// TIA Portal V17 export
// export: Created 2025-03-10T13:11:51.2223995Z, ExportSetting WithDefaults, DisplayName Totally Integrated Automation Portal, DisplayVersion V17 Update 8, DisplayName TIA Portal Openness, DisplayVersion V17 Update 8, DisplayName TIA Portal Version Control Interface, DisplayVersion V17, DisplayName SINAMICS Startdrive Advanced, DisplayVersion V17 SP2, DisplayName SINAMICS Startdrive G110M, G120, G120C, G120D, G120P, G115D, DisplayVersion V17 SP2, DisplayName SINAMICS Startdrive G130, G150, S120, S150, SINAMICS MV, S210, DisplayVersion V17 SP2, DisplayName STEP 7 Professional, DisplayVersion V17 Update 8, DisplayName SINUMERIK ONE STEP 7 Toolbox, DisplayVersion V17 Update 12, DisplayName SINUMERIK 840D sl STEP 7 Toolbox, DisplayVersion V17 Update 12, DisplayName STEP 7 Safety, DisplayVersion V17 Update 6, DisplayName WinCC Advanced, DisplayVersion V17 Update 8
VAR_GLOBAL   // PLC tag table "TAGS_IO_FIXTURES_UNIT_03"
   "/////MEASURING_UNIT/////" AT %M4500.0 : Bool;
   UMEAS_PUSHER_LCT_Q AT %M4500.1 : Bool;   // MEASURING UNIT LOCATE PUSHER OUTPUT
   UMEAS_PUSHER_RTN_Q AT %M4500.2 : Bool;   // MEASURING UNIT RETURN PUSHER OUTPUT
   UMEAS_PUSHER_UNLOCK_Q AT %M4500.3 : Bool;   // MEASURING UNIT UNLOCK PUSHER OUTPUT
   UMEAS_UNCLAMPED_I AT %M4500.4 : Bool;   // MEASURING UNIT PART UNCLAMPED INPUT
   UMEAS_CLAMPED_I AT %M4500.5 : Bool;   // MEASURING UNIT PART CLAMPED INPUT
   UMEAS_SPIN_CTRL_I AT %M4500.6 : Bool;   // MEASURING UNIT SPIN CONTROL INPUT
   UMEAS_PART_PRESENT_I AT %M4500.7 : Bool;   // MEASURING UNIT PART PRESENT INPUT
END_VAR
